Staubli VAL3: isSettled.pgx

public program isSettled(num& nSettled (dimensions=1))
  local bool bSettled
begin
  //robot moving = return 1/isSettled = false
  //robot stopped = return 0/isSettled = false
  bSettled=isSettled()
  switch bSettled
    case true
      nSettled=0
    break
    case false
      nSettled=1
    break
    default
      logMsg("error isSettled")
    break
  endSwitch
end
